(* IEC 61131-3 sources: RAG_PLC/data/result/test/034, 2 files *)

(* ---- wrapped.st ---- *)
(* =========================================================
   Generated by PLC-Eval Benchmark Wrapper
   ========================================================= *)

FUNCTION_BLOCK LLM_Wrapper_FB
VAR_INPUT
    N : INT;
    K : INT;
END_VAR

VAR_OUTPUT
    BINOM : INT;
END_VAR

VAR
    i : INT;
    N2 : INT;
    K2 : INT;
END_VAR

K2 := K;
N2 := N;
IF 2 * K2 > N2 THEN
    K2 := N2 - K2;
END_IF;
IF K2 > N2 THEN
    BINOM := 0;  // Return 0 if invalid input
ELSIF K2 = 0 OR K2 = N2 THEN
    BINOM := 1;
ELSIF K2 = 1 THEN
    BINOM := N2;
ELSE
    BINOM := N2;
    N2 := N2 + 1;
    FOR i := 2 TO K2 DO
        BINOM := BINOM * (N2 - i) / i;
    END_FOR;
END_IF;
END_FUNCTION_BLOCK

PROGRAM Auto_Proxy_Prg
  VAR
    instance : LLM_Wrapper_FB;
  END_VAR

  instance();
END_PROGRAM

CONFIGURATION Config0
  RESOURCE Res0 ON PLC
    TASK TaskMain(INTERVAL := T#20ms, PRIORITY := 0);
    PROGRAM Inst0 WITH TaskMain : Auto_Proxy_Prg;
  END_RESOURCE
END_CONFIGURATION

(* ---- raw_code.st ---- *)
VAR_INPUT
    N : INT;
    K : INT;
END_VAR

VAR_OUTPUT
    BINOM : INT;
END_VAR

VAR
    i : INT;
    N2 : INT;
    K2 : INT;
END_VAR

K2 := K;
N2 := N;
IF 2 * K2 > N2 THEN
    K2 := N2 - K2;
END_IF;
IF K2 > N2 THEN
    BINOM := 0;  // Return 0 if invalid input
ELSIF K2 = 0 OR K2 = N2 THEN
    BINOM := 1;
ELSIF K2 = 1 THEN
    BINOM := N2;
ELSE
    BINOM := N2;
    N2 := N2 + 1;
    FOR i := 2 TO K2 DO
        BINOM := BINOM * (N2 - i) / i;
    END_FOR;
END_IF;
